FUNCTION_BLOCK FB_HeatPumpSystem
VAR_INPUT
END_VAR
VAR
	PrimaryHeatpump: FB_Heatpump;
	HeatPumpInitTimeout: TON := (PT := TIME#3S0MS);
END_VAR

VAR_IN_OUT
	b_EnablePower 	: BOOL;
	//r_Setpoint 		: REAL;

//	Faults: ST_CoolingSystemEvents; 
//	HPSSet: ST_CoolingStackSet;
END_VAR

VAR_OUTPUT
	Get : ST_HeatpumpSystemGet;
END_VAR

VAR
	SecondHPPowerOnDelay: 	TON := (PT := TIME#250MS);
	IO	:	FB_HeatpumpSystem_IO;
	MBcommBusy	:	BOOL;
	CommFreeForID	:	BYTE	:= 0;
	CommFreeTimeout	:	TON 	:= (PT := TIME#5s0ms);
	SecondaryHeatPump: FB_Heatpump;
END_VAR

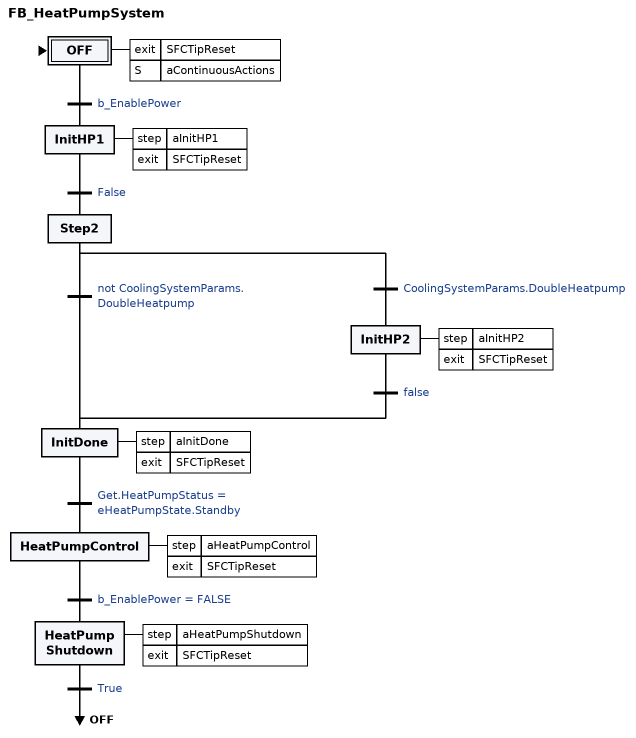
INITIAL_STEP OFF:
    SFCTipReset(P0);  // exit action
    aContinuousActions(S);
END_STEP
TRANSITION FROM OFF TO InitHP1
    := b_EnablePower;
END_TRANSITION
// macro InitHeatpumps begins
STEP InitHP1:
    aInitHP1(N);  // step action
    SFCTipReset(P0);  // exit action
END_STEP
TRANSITION FROM InitHP1 TO Step2
    := False;
END_TRANSITION
STEP Step2:
END_STEP
TRANSITION FROM Step2 TO InitDone
    := not CoolingSystemParams.DoubleHeatpump;
END_TRANSITION
TRANSITION FROM Step2 TO InitHP2
    := CoolingSystemParams.DoubleHeatpump;
END_TRANSITION
STEP InitHP2:
    aInitHP2(N);  // step action
    SFCTipReset(P0);  // exit action
END_STEP
TRANSITION FROM InitHP2 TO InitDone
    := false;
END_TRANSITION
STEP InitDone:
    aInitDone(N);  // step action
    SFCTipReset(P0);  // exit action
END_STEP
TRANSITION FROM InitDone TO HeatPumpControl
    := Get.HeatPumpStatus = eHeatPumpState.Standby;
END_TRANSITION
STEP HeatPumpControl:
    aHeatPumpControl(N);  // step action
    SFCTipReset(P0);  // exit action
END_STEP
TRANSITION FROM HeatPumpControl TO HeatPumpShutdown
    := b_EnablePower = FALSE;
END_TRANSITION
STEP HeatPumpShutdown:
    aHeatPumpShutdown(N);  // step action
    SFCTipReset(P0);  // exit action
END_STEP
TRANSITION FROM HeatPumpShutdown TO OFF
    := True;
END_TRANSITION

ACTION aContinuousActions:
IO(b_EnablePower := b_enablePower);

Get.PrimaryHeatpumpGet REF=PrimaryHeatPump.get;
Get.SecondaryHeatpumpGet REF=SecondaryHeatPump.get;

get.HeatPumpStatus := get.PrimaryHeatpumpGet.HeatPumpState;
END_ACTION

ACTION aHeatPumpControl:

//500ms trigger to switch MB bus ownership to next heatpump
CommFreeTimeout(in := NOT CommFreeTimeout.Q);
IF CommFreeTimeout.Q OR (not MBCommBusy) THEN
	CommFreeForID := (CommFreeForID+1) MOD 2;
END_IF

//FB returns MBCommBusy to indicate when status update is done. Could be used for optimized RW speed
//Not used at this moment

PrimaryHeatPump(ACPowerStatus := b_EnablePower, MBFree := (CommFreeForID=0), MBcommBusy => MBcommBusy);
//IF CoolingSystemParams.DoubleHeatpump THEN
//	HeatPumps[2](ACPowerStatus := b_EnablePower, MBFree := (CommFreeForID=1));
//END_IF
END_ACTION

ACTION aHeatPumpShutdown:
Get.HeatPumpStatus := eHeatPumpState.OFF;
END_ACTION

ACTION aInitDone:

get.HeatPumpStatus := eHeatPumpState.Standby;
END_ACTION

ACTION aInitHP1:

IF Coolingsystemparams.DoubleHeatpump THEN
	SecondaryHeatpump(ACPowerStatus := FALSE, MBFree := FALSE);
END_IF

IF PrimaryHeatpump.get.HeatPumpState <= eHeatpumpstate.Initializing THEN
	PrimaryHeatpump(ACPowerStatus := b_EnablePower, MBFree := TRUE);
ELSIF PrimaryHeatpump.get.HeatPumpState = eHeatpumpstate.Standby THEN
	PrimaryHeatpump(ACPowerStatus := b_EnablePower, MBFree := FALSE);
	SFCTip := TRUE;
END_IF
END_ACTION

ACTION aInitHP2:


IF SecondaryHeatpump.get.HeatPumpState = eHeatpumpstate.Initializing THEN
	SecondaryHeatpump(ACPowerStatus := b_EnablePower, MBFree := TRUE);
ELSIF SecondaryHeatpump.get.HeatPumpState = eHeatpumpstate.Standby THEN
	SecondaryHeatpump(ACPowerStatus := b_EnablePower, MBFree := FALSE);
	SFCTip := TRUE;
END_IF
END_ACTION

ACTION aPowerControl:
IO(b_EnablePower := b_enablePower);
END_ACTION

METHOD EMStop : BOOL
VAR_INPUT
END_VAR
EMstop := PrimaryHeatpump.emstop() and SecondaryHeatpump.emstop();
END_METHOD

METHOD GetDiagnostics 
VAR_IN_OUT
	AddError		: ARRAY [*] OF FB_AddErrorST;
	a_ActiveEvents	: ARRAY [*] OF ST_ErrorStruct;
	w_Index			: WORD;
END_VAR

VAR_OUTPUT
	b_errorActive	: BOOL;
	b_warningActive	: BOOL;
END_VAR

VAR
	by_errCt	: BYTE;
	by_warnCt	: BYTE;
	w_ID		: WORD;
END_VAR

//check if this call works:
PrimaryHeatpump.GetDiagnostics(AddError := AddError, a_ActiveEvents := a_ActiveEvents, w_Index := w_Index, b_errorActive => b_errorActive, b_warningActive => b_warningActive);

//not in use
//Heatpumps[2].GetDiagnostics(AddError := AddError, a_ActiveEvents := a_ActiveEvents, w_Index := w_Index, b_errorActive => b_errorActive, b_warningActive => b_warningActive);
END_METHOD

METHOD Reset : BOOL
VAR_INPUT
END_VAR
Reset := PrimaryHeatpump.Reset() and SecondaryHeatpump.Reset();
END_METHOD

ACTION SFCTipReset:
SFCTip := FALSE;
END_ACTION

METHOD WriteSetpoint : BOOL
VAR_INPUT
	OperatingMode	:	eHeatpumpMode;
	SetPoint		: 	REAL;
END_VAR
PrimaryHeatpump.WriteSetpoint(OperatingMode := OperatingMode, SetPoint := Setpoint);

//This method will also contain potential master/slave temperature differentials and other differences between heatpumps
//Heatpumps[2].WriteSetpoint(OperatingMode := OperatingMode);
END_METHOD

END_FUNCTION_BLOCK

(* stored: Version 1.1.0.1, ProductVersion 3.1.4024.12
   POU FB_HeatPumpSystem: Id {fd3ced53-38d6-4a15-8e68-1fb19bd16ace}, SpecialFunc None
   Folder InternalActions: Id {c20474ff-e84c-47d0-8534-715ec07a3b59}
   Action aContinuousActions: Id {16e92865-ea65-42fa-be94-fa3158d56caf}
   Action aHeatPumpControl: Id {40cb6c99-f2bd-4463-aec6-f0b22d5ed475}
   Action aHeatPumpShutdown: Id {dfa77b7c-2af9-473e-b37e-15d67f751833}
   Action aInitDone: Id {e06a6405-dcf9-4ae4-bfbe-c27fe02a41f7}
   Action aInitHP1: Id {1d819cdb-f81a-426e-9213-238391d386d3}
   Action aInitHP2: Id {594411e8-2bfb-4a64-a290-320fec4b45d8}
   Action aPowerControl: Id {7a742825-0880-4e7a-b565-fd6af40350f5}
   Method EMStop: Id {c5d59058-fc75-4523-8e14-2a1384499863}
   Method GetDiagnostics: Id {897c308b-8471-40f4-850e-e89d0aac515c}
   Method Reset: Id {4a0bb0ee-0ec3-4295-bbf7-b62e6e6a1cef}
   Action SFCTipReset: Id {eb10d883-3ce0-4bca-9d41-17668d540ab5}
   Method WriteSetpoint: Id {18c61e5f-7dfc-42d9-af3e-d11734e33e5d} *)
